//==================================================================================================
//								RJM Maszyny sp. z o.o.
//									04.02.2022
//	Obsługa elektrozaworu 3/2 normalnie otwartego
// 	v1.0	|| TC v 3.1.4024.22		|| - pierwsza wersja
//==================================================================================================
FUNCTION_BLOCK FB_Elektrozawor_3na2_NO implements I_Elektrozawor_3na2
VAR
	fbCewka									: FB_ElektrozaworCewka;
END_VAR

//==================================================================================================
//								RJM Maszyny sp. z o.o.
//									04.02.2022
//	Włączenie cewki - wyjscie 2
// 	v1.0	|| TC v 3.1.4024.22		|| - pierwsza wersja
//==================================================================================================
METHOD Wlacz
VAR_INPUT
END_VAR
fbCewka.Wlacz ();
END_METHOD

//==================================================================================================
//								RJM Maszyny sp. z o.o.
//									04.02.2022
//	Wyłączenie cewki - wyjscie 2
// 	v1.0	|| TC v 3.1.4024.22		|| - pierwsza wersja
//==================================================================================================
METHOD Wylacz
VAR_INPUT
END_VAR
fbCewka.Wylacz ();
END_METHOD

END_FUNCTION_BLOCK

(* stored: Version 1.1.0.1, ProductVersion 3.1.4024.11
   POU FB_Elektrozawor_3na2_NO: Id {a76f145e-398d-4fed-98d7-f3ef1af1e802}, SpecialFunc None
   Method Wlacz: Id {27c4f4fd-ed0e-46b0-9b2e-bd9454e7f642}
   Method Wylacz: Id {317c732e-5820-4268-89c3-f41fc27c4b76} *)
